// TIA Portal V17 export
// export: Created 2023-03-06T02:05:17.8449285Z, ExportSetting WithDefaults, DisplayName Totally Integrated Automation Portal, DisplayVersion V17 Update 4, DisplayName TIA Portal Openness, DisplayVersion V17 Update 4, DisplayName TIA Portal Version Control Interface, DisplayVersion V17, DisplayName STEP 7 Professional, DisplayVersion V17 Update 4, DisplayName STEP 7 Safety, DisplayVersion V17, DisplayName WinCC Professional, DisplayVersion V17 Update 4
DATA_BLOCK "DashBoard"   // DB121
{ S7_Optimized_Access := 'FALSE' }
VERSION : 0.1
// stored: AutoNumber false, DBAccessibleFromOPCUA true, DBAccessibleFromWebserver true, IsOnlyStoredInLoadMemory false, IsWriteProtectedInAS false
   VAR
      BB1 { S7_SetPoint := 'True'} : "BB";
      BB2 { S7_SetPoint := 'True'} : "BB";
      BB1BR1 : "BR";
      BB1BR2 : "BR";
      BB1BR3 : "BR";
      BB1BR4 : "BR";
      BB1BR5 : "BR";
      BB1BR6 : "BR";
      BB1BR7 : "BR";
      BB1BR8 : "BR";
      BB1BR9 : "BR";
      BB1BR10 : "BR";
      BB1BR11 : "BR";
      BB1BR12 : "BR";
      BB2BR1 : "BR";
      BB2BR2 : "BR";
      BB2BR3 : "BR";
      BB2BR4 : "BR";
      BB2BR5 : "BR";
      BB2BR6 : "BR";
      BB2BR7 : "BR";
      BB2BR8 : "BR";
      BB2BR9 : "BR";
      BB2BR10 : "BR";
      BB2BR11 : "BR";
      BB2BR12 : "BR";
      PCS : "PCS";
      MVSKID { S7_SetPoint := 'True'} : "MVSKID";
      SM { S7_SetPoint := 'True'} : "SM";
   END_VAR
BEGIN
END_DATA_BLOCK
